Universal Robots PolyScope program: tmp_water.urp

Program tmp_water (installation=20240827 directory=/programs/show createdIn=5.15.1 lastSavedIn=5.15.1 robotSerialNumber=20245500285)
Calibrated DH parameters: a=[0.000097, -0.210459, -0.026602, 0.000137, 0.000078, 0]; d=[0.162601, 254.180657, -54.076236, -199.970743, 0.099615, 0.099684]; alpha=[1.569796, -0.001455, 0.001957, 1.570525, -1.571561, 0]; deltaTheta=[0, -1.053331, 8.839472, -1.50296, 0.000002, 0]
InitVariablesNode
Robot Program (runOnlyOnce=false)
  Script: usb = rpc_factory("xmlrpc","http://192.168.1.7:9120/RPC2")
  Script: usb.open()
  Popup Message (haltProgram=false message=1 inputType=Text)
  pos := 30.86
  Script: usb.close( True ,pos)
  Popup Message (haltProgram=false message=1 inputType=Text)
  '1'
  Wait Sleep waitTime=6.15
  pos := pos+1
  Script: usb.close( True ,pos)
  '2'
  Wait Sleep waitTime=0.05
  pos := pos+1
  Script: usb.close( True ,pos)
  '3'
  Wait Sleep waitTime=0.05
  pos := pos+1
  Script: usb.close( True ,pos)
  '4'
  Wait Sleep waitTime=0.41
  pos := pos+1
  Script: usb.close( True ,pos)
  '5'
  Wait Sleep waitTime=0.66
  pos := pos+1
  Script: usb.close( True ,pos)
  '6'
  Wait Sleep waitTime=0.04
  pos := pos+1
  Script: usb.close( True ,pos)
  '7'
  Wait Sleep waitTime=2.12
  pos := pos+1
  Script: usb.close( True ,pos)
  '8'
  Wait Sleep waitTime=2.57
  Popup Message (haltProgram=false message=1 inputType=Text)
  pos := pos+1
  Script: usb.close( True ,pos)
  '9'
  Wait Sleep waitTime=0.04
  pos := pos+1
  Script: usb.close( True ,pos)
  '10'
  Wait Sleep waitTime=0.34
  pos := pos+1
  Script: usb.close( True ,pos)
  Popup Message (haltProgram=false message=2 inputType=Text)
